// TIA Portal project "P1" (V17)

(* hardware
DEVICE "S7-1500/ET200MP station_1"  S7-1500 station
   slot 0: "Rail_0"  Rack  6ES7 590-1***0-0AA0
   slot 1: "PLC_1"  CPU 1513-1 PN  6ES7 513-1AL00-0AB0  V1.8
      slot 3: "CPU display_1"  6ES7591-1AA00-0AA0
      slot 32768: "PROFINET interface_1"  X1
         slot 32769: "Port_1"  X1 P1
         slot 32770: "Port_2"  X1 P2
*)

// ===== PLC "PLC_1"  CPU 1513-1 PN =====

VAR_GLOBAL   // PLC tag table "Default tag table"
   "INT" AT %MW100 : Int;   // Analog value from the temp controller
   "DINT" AT %MD104 : DInt;   // Actual value from the temp controller
   "MULTIPLICACION" AT %MD108 : DInt;   // Multiplicacion
   "ACTUAL" AT %MD112 : DInt;   // Actual Temperatura IN (°C)
END_VAR

ORGANIZATION_BLOCK "Main"   // OB1, LAD, ProgramCycle
TITLE = "Main Program Sweep (Cycle)"
{ S7_Optimized_Access := 'TRUE' }
VERSION : 0.1
// Esta configuracion, Utilizamos un controlador de temp conectado a un sensor RTD que mide la temperatura de un tanque. El controlador emite una señal analogica de 0-10 V CC proporcionala la temperatura medida (0 - 100 °C) Esta señal analogica es leida por un PLC (SIEMENS) procesada y convertida a la temperatura Real en grados celsius utilizando la logica de escalera estructurada.
   VAR_INPUT
      Initial_Call : Bool;   // Initial call of this OB
      Remanence : Bool;   // =True, if remanent data are available
   END_VAR
BEGIN

REGION Network 1: Convertir valor de INT a DINT
   // Entrada %MW100 (Registro de entrada Analogica)
   // Salida %MD104 (Valor DINT para mas matematicas)
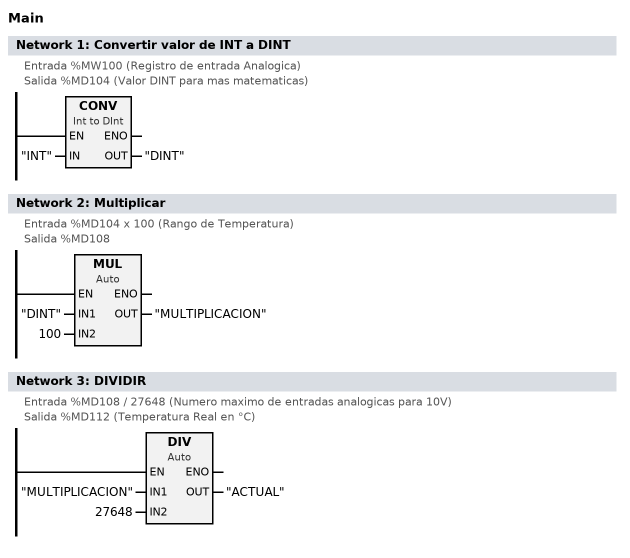
   RUNG wire#powerrail
      { S7_Templates := "[SrcType := Int, DestType := DInt]" } Convert(in := "INT", out => "DINT")
   END_RUNG
   // the same network as SCL:
   "DINT" := INT_TO_DINT("INT");
END_REGION

REGION Network 2: Multiplicar
   // Entrada %MD104 x 100 (Rango de Temperatura)
   // Salida %MD108
   RUNG wire#powerrail
      Mul(in1 := "DINT", in2 := 100, out => "MULTIPLICACION")
   END_RUNG
   // the same network as SCL:
   "MULTIPLICACION" := "DINT" * 100;
END_REGION

REGION Network 3: DIVIDIR
   // Entrada %MD108 / 27648 (Numero maximo de entradas analogicas para 10V)
   // Salida %MD112 (Temperatura Real en °C)
   RUNG wire#powerrail
      Div(in1 := "MULTIPLICACION", in2 := 27648, out => "ACTUAL")
   END_RUNG
   // the same network as SCL:
   "ACTUAL" := "MULTIPLICACION" / 27648;
END_REGION
END_ORGANIZATION_BLOCK